ABB RAPID module: etna.mod

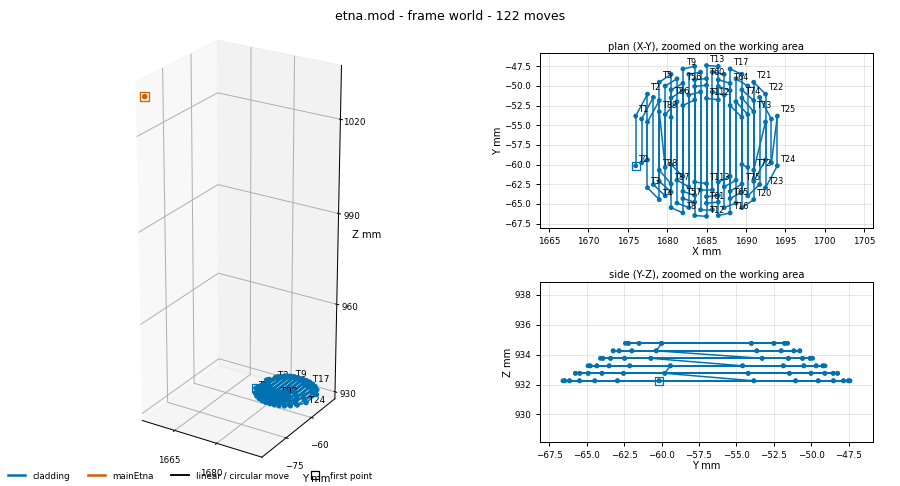
[picture p0: tool path of etna.mod in frame world, 122 of 122 moves have a stored position in this frame; points joined in program order, loops and branches not executed]
MODULE Etna

    PERS tooldata toolEtna:=[TRUE,[[215.7,-22.4,473.8],[0.500000,0.000000,-0.866025,0.000000]],[20,[70,30,123.5],[0,0,1,0],1,0,1]];
    PERS wobjdata wobjEtna:=[FALSE,TRUE,"",[[1655.0,-87.0,932.0],[1.000000,0.000000,0.000000,0.000000]],[[0,0,0],[1,0,0,0]]];

    VAR triggdata laserON;
    VAR triggdata laserOFF;

    CONST speeddata vl:=[8,500,5000,1000];


    CONST robtarget T0:=[[21.000000,26.839411,0.250000],[1.000000,0.000000,0.000000,0.000000],[-1,0,-1,0],[9E+09,9E+09,9E+09,9E+09,9E+09,9E+09]];
    CONST robtarget T1:=[[21.000000,33.160593,0.250000],[1.000000,0.000000,0.000000,0.000000],[-1,0,-1,0],[9E+09,9E+09,9E+09,9E+09,9E+09,9E+09]];
    CONST robtarget T2:=[[22.500000,35.946596,0.250000],[1.000000,0.000000,0.000000,0.000000],[-1,0,-1,0],[9E+09,9E+09,9E+09,9E+09,9E+09,9E+09]];
    CONST robtarget T3:=[[22.500000,24.053408,0.250000],[1.000000,0.000000,0.000000,0.000000],[-1,0,-1,0],[9E+09,9E+09,9E+09,9E+09,9E+09,9E+09]];
    CONST robtarget T4:=[[24.000000,22.537615,0.250000],[1.000000,0.000000,0.000000,0.000000],[-1,0,-1,0],[9E+09,9E+09,9E+09,9E+09,9E+09,9E+09]];
    CONST robtarget T5:=[[24.000000,37.462389,0.250000],[1.000000,0.000000,0.000000,0.000000],[-1,0,-1,0],[9E+09,9E+09,9E+09,9E+09,9E+09,9E+09]];
    CONST robtarget T6:=[[25.500000,38.475702,0.250000],[1.000000,0.000000,0.000000,0.000000],[-1,0,-1,0],[9E+09,9E+09,9E+09,9E+09,9E+09,9E+09]];
    CONST robtarget T7:=[[25.500000,21.524301,0.250000],[1.000000,0.000000,0.000000,0.000000],[-1,0,-1,0],[9E+09,9E+09,9E+09,9E+09,9E+09,9E+09]];
    CONST robtarget T8:=[[27.000000,20.852779,0.250000],[1.000000,0.000000,0.000000,0.000000],[-1,0,-1,0],[9E+09,9E+09,9E+09,9E+09,9E+09,9E+09]];
    CONST robtarget T9:=[[27.000000,39.147225,0.250000],[1.000000,0.000000,0.000000,0.000000],[-1,0,-1,0],[9E+09,9E+09,9E+09,9E+09,9E+09,9E+09]];
    CONST robtarget T10:=[[28.500000,39.476842,0.250000],[1.000000,0.000000,0.000000,0.000000],[-1,0,-1,0],[9E+09,9E+09,9E+09,9E+09,9E+09,9E+09]];
    CONST robtarget T11:=[[28.500000,20.523160,0.250000],[1.000000,0.000000,0.000000,0.000000],[-1,0,-1,0],[9E+09,9E+09,9E+09,9E+09,9E+09,9E+09]];
    CONST robtarget T12:=[[30.000000,20.416667,0.250000],[1.000000,0.000000,0.000000,0.000000],[-1,0,-1,0],[9E+09,9E+09,9E+09,9E+09,9E+09,9E+09]];
    CONST robtarget T13:=[[30.000000,39.583335,0.250000],[1.000000,0.000000,0.000000,0.000000],[-1,0,-1,0],[9E+09,9E+09,9E+09,9E+09,9E+09,9E+09]];
    CONST robtarget T14:=[[31.500000,39.476842,0.250000],[1.000000,0.000000,0.000000,0.000000],[-1,0,-1,0],[9E+09,9E+09,9E+09,9E+09,9E+09,9E+09]];
    CONST robtarget T15:=[[31.500000,20.523161,0.250000],[1.000000,0.000000,0.000000,0.000000],[-1,0,-1,0],[9E+09,9E+09,9E+09,9E+09,9E+09,9E+09]];
    CONST robtarget T16:=[[33.000000,20.852779,0.250000],[1.000000,0.000000,0.000000,0.000000],[-1,0,-1,0],[9E+09,9E+09,9E+09,9E+09,9E+09,9E+09]];
    CONST robtarget T17:=[[33.000000,39.147225,0.250000],[1.000000,0.000000,0.000000,0.000000],[-1,0,-1,0],[9E+09,9E+09,9E+09,9E+09,9E+09,9E+09]];
    CONST robtarget T18:=[[34.500000,38.475702,0.250000],[1.000000,0.000000,0.000000,0.000000],[-1,0,-1,0],[9E+09,9E+09,9E+09,9E+09,9E+09,9E+09]];
    CONST robtarget T19:=[[34.500000,21.524301,0.250000],[1.000000,0.000000,0.000000,0.000000],[-1,0,-1,0],[9E+09,9E+09,9E+09,9E+09,9E+09,9E+09]];
    CONST robtarget T20:=[[36.000000,22.537615,0.250000],[1.000000,0.000000,0.000000,0.000000],[-1,0,-1,0],[9E+09,9E+09,9E+09,9E+09,9E+09,9E+09]];
    CONST robtarget T21:=[[36.000000,37.462389,0.250000],[1.000000,0.000000,0.000000,0.000000],[-1,0,-1,0],[9E+09,9E+09,9E+09,9E+09,9E+09,9E+09]];
    CONST robtarget T22:=[[37.500000,35.946596,0.250000],[1.000000,0.000000,0.000000,0.000000],[-1,0,-1,0],[9E+09,9E+09,9E+09,9E+09,9E+09,9E+09]];
    CONST robtarget T23:=[[37.500000,24.053407,0.250000],[1.000000,0.000000,0.000000,0.000000],[-1,0,-1,0],[9E+09,9E+09,9E+09,9E+09,9E+09,9E+09]];
    CONST robtarget T24:=[[39.000000,26.839410,0.250000],[1.000000,0.000000,0.000000,0.000000],[-1,0,-1,0],[9E+09,9E+09,9E+09,9E+09,9E+09,9E+09]];
    CONST robtarget T25:=[[39.000000,33.160593,0.250000],[1.000000,0.000000,0.000000,0.000000],[-1,0,-1,0],[9E+09,9E+09,9E+09,9E+09,9E+09,9E+09]];
    CONST robtarget T26:=[[38.250000,27.215156,0.750000],[1.000000,0.000000,0.000000,0.000000],[-1,0,-1,0],[9E+09,9E+09,9E+09,9E+09,9E+09,9E+09]];
    CONST robtarget T27:=[[38.250000,32.784847,0.750000],[1.000000,0.000000,0.000000,0.000000],[-1,0,-1,0],[9E+09,9E+09,9E+09,9E+09,9E+09,9E+09]];
    CONST robtarget T28:=[[36.750000,35.538746,0.750000],[1.000000,0.000000,0.000000,0.000000],[-1,0,-1,0],[9E+09,9E+09,9E+09,9E+09,9E+09,9E+09]];
    CONST robtarget T29:=[[36.750000,24.461257,0.750000],[1.000000,0.000000,0.000000,0.000000],[-1,0,-1,0],[9E+09,9E+09,9E+09,9E+09,9E+09,9E+09]];
    CONST robtarget T30:=[[35.250000,23.019764,0.750000],[1.000000,0.000000,0.000000,0.000000],[-1,0,-1,0],[9E+09,9E+09,9E+09,9E+09,9E+09,9E+09]];
    CONST robtarget T31:=[[35.250000,36.980240,0.750000],[1.000000,0.000000,0.000000,0.000000],[-1,0,-1,0],[9E+09,9E+09,9E+09,9E+09,9E+09,9E+09]];
    CONST robtarget T32:=[[33.750000,37.899267,0.750000],[1.000000,0.000000,0.000000,0.000000],[-1,0,-1,0],[9E+09,9E+09,9E+09,9E+09,9E+09,9E+09]];
    CONST robtarget T33:=[[33.750000,22.100737,0.750000],[1.000000,0.000000,0.000000,0.000000],[-1,0,-1,0],[9E+09,9E+09,9E+09,9E+09,9E+09,9E+09]];
    CONST robtarget T34:=[[32.250000,21.535407,0.750000],[1.000000,0.000000,0.000000,0.000000],[-1,0,-1,0],[9E+09,9E+09,9E+09,9E+09,9E+09,9E+09]];
    CONST robtarget T35:=[[32.250000,38.464597,0.750000],[1.000000,0.000000,0.000000,0.000000],[-1,0,-1,0],[9E+09,9E+09,9E+09,9E+09,9E+09,9E+09]];
    CONST robtarget T36:=[[30.750000,38.750002,0.750000],[1.000000,0.000000,0.000000,0.000000],[-1,0,-1,0],[9E+09,9E+09,9E+09,9E+09,9E+09,9E+09]];
    CONST robtarget T37:=[[30.750000,21.250000,0.750000],[1.000000,0.000000,0.000000,0.000000],[-1,0,-1,0],[9E+09,9E+09,9E+09,9E+09,9E+09,9E+09]];
    CONST robtarget T38:=[[29.250000,21.250000,0.750000],[1.000000,0.000000,0.000000,0.000000],[-1,0,-1,0],[9E+09,9E+09,9E+09,9E+09,9E+09,9E+09]];
    CONST robtarget T39:=[[29.250000,38.750002,0.750000],[1.000000,0.000000,0.000000,0.000000],[-1,0,-1,0],[9E+09,9E+09,9E+09,9E+09,9E+09,9E+09]];
    CONST robtarget T40:=[[27.750000,38.464597,0.750000],[1.000000,0.000000,0.000000,0.000000],[-1,0,-1,0],[9E+09,9E+09,9E+09,9E+09,9E+09,9E+09]];
    CONST robtarget T41:=[[27.750000,21.535406,0.750000],[1.000000,0.000000,0.000000,0.000000],[-1,0,-1,0],[9E+09,9E+09,9E+09,9E+09,9E+09,9E+09]];
    CONST robtarget T42:=[[26.250000,22.100737,0.750000],[1.000000,0.000000,0.000000,0.000000],[-1,0,-1,0],[9E+09,9E+09,9E+09,9E+09,9E+09,9E+09]];
    CONST robtarget T43:=[[26.250000,37.899267,0.750000],[1.000000,0.000000,0.000000,0.000000],[-1,0,-1,0],[9E+09,9E+09,9E+09,9E+09,9E+09,9E+09]];
    CONST robtarget T44:=[[24.750000,36.980240,0.750000],[1.000000,0.000000,0.000000,0.000000],[-1,0,-1,0],[9E+09,9E+09,9E+09,9E+09,9E+09,9E+09]];
    CONST robtarget T45:=[[24.750000,23.019764,0.750000],[1.000000,0.000000,0.000000,0.000000],[-1,0,-1,0],[9E+09,9E+09,9E+09,9E+09,9E+09,9E+09]];
    CONST robtarget T46:=[[23.250000,24.461257,0.750000],[1.000000,0.000000,0.000000,0.000000],[-1,0,-1,0],[9E+09,9E+09,9E+09,9E+09,9E+09,9E+09]];
    CONST robtarget T47:=[[23.250000,35.538747,0.750000],[1.000000,0.000000,0.000000,0.000000],[-1,0,-1,0],[9E+09,9E+09,9E+09,9E+09,9E+09,9E+09]];
    CONST robtarget T48:=[[21.750000,32.784848,0.750000],[1.000000,0.000000,0.000000,0.000000],[-1,0,-1,0],[9E+09,9E+09,9E+09,9E+09,9E+09,9E+09]];
    CONST robtarget T49:=[[21.750000,27.215157,0.750000],[1.000000,0.000000,0.000000,0.000000],[-1,0,-1,0],[9E+09,9E+09,9E+09,9E+09,9E+09,9E+09]];
    CONST robtarget T50:=[[22.500000,27.590903,1.250000],[1.000000,0.000000,0.000000,0.000000],[-1,0,-1,0],[9E+09,9E+09,9E+09,9E+09,9E+09,9E+09]];
    CONST robtarget T51:=[[22.500000,32.409103,1.250000],[1.000000,0.000000,0.000000,0.000000],[-1,0,-1,0],[9E+09,9E+09,9E+09,9E+09,9E+09,9E+09]];
    CONST robtarget T52:=[[24.000000,35.130897,1.250000],[1.000000,0.000000,0.000000,0.000000],[-1,0,-1,0],[9E+09,9E+09,9E+09,9E+09,9E+09,9E+09]];
    CONST robtarget T53:=[[24.000000,24.869107,1.250000],[1.000000,0.000000,0.000000,0.000000],[-1,0,-1,0],[9E+09,9E+09,9E+09,9E+09,9E+09,9E+09]];
    CONST robtarget T54:=[[25.500000,23.501912,1.250000],[1.000000,0.000000,0.000000,0.000000],[-1,0,-1,0],[9E+09,9E+09,9E+09,9E+09,9E+09,9E+09]];
    CONST robtarget T55:=[[25.500000,36.498092,1.250000],[1.000000,0.000000,0.000000,0.000000],[-1,0,-1,0],[9E+09,9E+09,9E+09,9E+09,9E+09,9E+09]];
    CONST robtarget T56:=[[27.000000,37.322831,1.250000],[1.000000,0.000000,0.000000,0.000000],[-1,0,-1,0],[9E+09,9E+09,9E+09,9E+09,9E+09,9E+09]];
    CONST robtarget T57:=[[27.000000,22.677173,1.250000],[1.000000,0.000000,0.000000,0.000000],[-1,0,-1,0],[9E+09,9E+09,9E+09,9E+09,9E+09,9E+09]];
    CONST robtarget T58:=[[28.500000,22.227061,1.250000],[1.000000,0.000000,0.000000,0.000000],[-1,0,-1,0],[9E+09,9E+09,9E+09,9E+09,9E+09,9E+09]];
    CONST robtarget T59:=[[28.500000,37.772941,1.250000],[1.000000,0.000000,0.000000,0.000000],[-1,0,-1,0],[9E+09,9E+09,9E+09,9E+09,9E+09,9E+09]];
    CONST robtarget T60:=[[30.000000,37.916669,1.250000],[1.000000,0.000000,0.000000,0.000000],[-1,0,-1,0],[9E+09,9E+09,9E+09,9E+09,9E+09,9E+09]];
    CONST robtarget T61:=[[30.000000,22.083334,1.250000],[1.000000,0.000000,0.000000,0.000000],[-1,0,-1,0],[9E+09,9E+09,9E+09,9E+09,9E+09,9E+09]];
    CONST robtarget T62:=[[31.500000,22.227062,1.250000],[1.000000,0.000000,0.000000,0.000000],[-1,0,-1,0],[9E+09,9E+09,9E+09,9E+09,9E+09,9E+09]];
    CONST robtarget T63:=[[31.500000,37.772942,1.250000],[1.000000,0.000000,0.000000,0.000000],[-1,0,-1,0],[9E+09,9E+09,9E+09,9E+09,9E+09,9E+09]];
    CONST robtarget T64:=[[33.000000,37.322831,1.250000],[1.000000,0.000000,0.000000,0.000000],[-1,0,-1,0],[9E+09,9E+09,9E+09,9E+09,9E+09,9E+09]];
    CONST robtarget T65:=[[33.000000,22.677173,1.250000],[1.000000,0.000000,0.000000,0.000000],[-1,0,-1,0],[9E+09,9E+09,9E+09,9E+09,9E+09,9E+09]];
    CONST robtarget T66:=[[34.500000,23.501912,1.250000],[1.000000,0.000000,0.000000,0.000000],[-1,0,-1,0],[9E+09,9E+09,9E+09,9E+09,9E+09,9E+09]];
    CONST robtarget T67:=[[34.500000,36.498092,1.250000],[1.000000,0.000000,0.000000,0.000000],[-1,0,-1,0],[9E+09,9E+09,9E+09,9E+09,9E+09,9E+09]];
    CONST robtarget T68:=[[36.000000,35.130896,1.250000],[1.000000,0.000000,0.000000,0.000000],[-1,0,-1,0],[9E+09,9E+09,9E+09,9E+09,9E+09,9E+09]];
    CONST robtarget T69:=[[36.000000,24.869107,1.250000],[1.000000,0.000000,0.000000,0.000000],[-1,0,-1,0],[9E+09,9E+09,9E+09,9E+09,9E+09,9E+09]];
    CONST robtarget T70:=[[37.500000,27.590901,1.250000],[1.000000,0.000000,0.000000,0.000000],[-1,0,-1,0],[9E+09,9E+09,9E+09,9E+09,9E+09,9E+09]];
    CONST robtarget T71:=[[37.500000,32.409101,1.250000],[1.000000,0.000000,0.000000,0.000000],[-1,0,-1,0],[9E+09,9E+09,9E+09,9E+09,9E+09,9E+09]];
    CONST robtarget T72:=[[36.000000,26.282882,1.750000],[1.000000,0.000000,0.000000,0.000000],[-1,0,-1,0],[9E+09,9E+09,9E+09,9E+09,9E+09,9E+09]];
    CONST robtarget T73:=[[36.000000,33.717123,1.750000],[1.000000,0.000000,0.000000,0.000000],[-1,0,-1,0],[9E+09,9E+09,9E+09,9E+09,9E+09,9E+09]];
    CONST robtarget T74:=[[34.500000,35.468036,1.750000],[1.000000,0.000000,0.000000,0.000000],[-1,0,-1,0],[9E+09,9E+09,9E+09,9E+09,9E+09,9E+09]];
    CONST robtarget T75:=[[34.500000,24.531968,1.750000],[1.000000,0.000000,0.000000,0.000000],[-1,0,-1,0],[9E+09,9E+09,9E+09,9E+09,9E+09,9E+09]];
    CONST robtarget T76:=[[33.000000,23.589370,1.750000],[1.000000,0.000000,0.000000,0.000000],[-1,0,-1,0],[9E+09,9E+09,9E+09,9E+09,9E+09,9E+09]];
    CONST robtarget T77:=[[33.000000,36.410634,1.750000],[1.000000,0.000000,0.000000,0.000000],[-1,0,-1,0],[9E+09,9E+09,9E+09,9E+09,9E+09,9E+09]];
    CONST robtarget T78:=[[31.500000,36.920992,1.750000],[1.000000,0.000000,0.000000,0.000000],[-1,0,-1,0],[9E+09,9E+09,9E+09,9E+09,9E+09,9E+09]];
    CONST robtarget T79:=[[31.500000,23.079013,1.750000],[1.000000,0.000000,0.000000,0.000000],[-1,0,-1,0],[9E+09,9E+09,9E+09,9E+09,9E+09,9E+09]];
    CONST robtarget T80:=[[30.000000,22.916668,1.750000],[1.000000,0.000000,0.000000,0.000000],[-1,0,-1,0],[9E+09,9E+09,9E+09,9E+09,9E+09,9E+09]];
    CONST robtarget T81:=[[30.000000,37.083335,1.750000],[1.000000,0.000000,0.000000,0.000000],[-1,0,-1,0],[9E+09,9E+09,9E+09,9E+09,9E+09,9E+09]];
    CONST robtarget T82:=[[28.500000,36.920991,1.750000],[1.000000,0.000000,0.000000,0.000000],[-1,0,-1,0],[9E+09,9E+09,9E+09,9E+09,9E+09,9E+09]];
    CONST robtarget T83:=[[28.500000,23.079011,1.750000],[1.000000,0.000000,0.000000,0.000000],[-1,0,-1,0],[9E+09,9E+09,9E+09,9E+09,9E+09,9E+09]];
    CONST robtarget T84:=[[27.000000,23.589370,1.750000],[1.000000,0.000000,0.000000,0.000000],[-1,0,-1,0],[9E+09,9E+09,9E+09,9E+09,9E+09,9E+09]];
    CONST robtarget T85:=[[27.000000,36.410634,1.750000],[1.000000,0.000000,0.000000,0.000000],[-1,0,-1,0],[9E+09,9E+09,9E+09,9E+09,9E+09,9E+09]];
    CONST robtarget T86:=[[25.500000,35.468036,1.750000],[1.000000,0.000000,0.000000,0.000000],[-1,0,-1,0],[9E+09,9E+09,9E+09,9E+09,9E+09,9E+09]];
    CONST robtarget T87:=[[25.500000,24.531968,1.750000],[1.000000,0.000000,0.000000,0.000000],[-1,0,-1,0],[9E+09,9E+09,9E+09,9E+09,9E+09,9E+09]];
    CONST robtarget T88:=[[24.000000,26.282881,1.750000],[1.000000,0.000000,0.000000,0.000000],[-1,0,-1,0],[9E+09,9E+09,9E+09,9E+09,9E+09,9E+09]];
    CONST robtarget T89:=[[24.000000,33.717121,1.750000],[1.000000,0.000000,0.000000,0.000000],[-1,0,-1,0],[9E+09,9E+09,9E+09,9E+09,9E+09,9E+09]];
    CONST robtarget T90:=[[24.750000,26.643354,2.250000],[1.000000,0.000000,0.000000,0.000000],[-1,0,-1,0],[9E+09,9E+09,9E+09,9E+09,9E+09,9E+09]];
    CONST robtarget T91:=[[24.750000,33.356648,2.250000],[1.000000,0.000000,0.000000,0.000000],[-1,0,-1,0],[9E+09,9E+09,9E+09,9E+09,9E+09,9E+09]];
    CONST robtarget T92:=[[26.250000,34.985887,2.250000],[1.000000,0.000000,0.000000,0.000000],[-1,0,-1,0],[9E+09,9E+09,9E+09,9E+09,9E+09,9E+09]];
    CONST robtarget T93:=[[26.250000,25.014116,2.250000],[1.000000,0.000000,0.000000,0.000000],[-1,0,-1,0],[9E+09,9E+09,9E+09,9E+09,9E+09,9E+09]];
    CONST robtarget T94:=[[27.750000,24.165805,2.250000],[1.000000,0.000000,0.000000,0.000000],[-1,0,-1,0],[9E+09,9E+09,9E+09,9E+09,9E+09,9E+09]];
    CONST robtarget T95:=[[27.750000,35.834199,2.250000],[1.000000,0.000000,0.000000,0.000000],[-1,0,-1,0],[9E+09,9E+09,9E+09,9E+09,9E+09,9E+09]];
    CONST robtarget T96:=[[29.250000,36.229335,2.250000],[1.000000,0.000000,0.000000,0.000000],[-1,0,-1,0],[9E+09,9E+09,9E+09,9E+09,9E+09,9E+09]];
    CONST robtarget T97:=[[29.250000,23.770668,2.250000],[1.000000,0.000000,0.000000,0.000000],[-1,0,-1,0],[9E+09,9E+09,9E+09,9E+09,9E+09,9E+09]];
    CONST robtarget T98:=[[30.750000,23.770668,2.250000],[1.000000,0.000000,0.000000,0.000000],[-1,0,-1,0],[9E+09,9E+09,9E+09,9E+09,9E+09,9E+09]];
    CONST robtarget T99:=[[30.750000,36.229335,2.250000],[1.000000,0.000000,0.000000,0.000000],[-1,0,-1,0],[9E+09,9E+09,9E+09,9E+09,9E+09,9E+09]];
    CONST robtarget T100:=[[32.250000,35.834199,2.250000],[1.000000,0.000000,0.000000,0.000000],[-1,0,-1,0],[9E+09,9E+09,9E+09,9E+09,9E+09,9E+09]];
    CONST robtarget T101:=[[32.250000,24.165805,2.250000],[1.000000,0.000000,0.000000,0.000000],[-1,0,-1,0],[9E+09,9E+09,9E+09,9E+09,9E+09,9E+09]];
    CONST robtarget T102:=[[33.750000,25.014116,2.250000],[1.000000,0.000000,0.000000,0.000000],[-1,0,-1,0],[9E+09,9E+09,9E+09,9E+09,9E+09,9E+09]];
    CONST robtarget T103:=[[33.750000,34.985887,2.250000],[1.000000,0.000000,0.000000,0.000000],[-1,0,-1,0],[9E+09,9E+09,9E+09,9E+09,9E+09,9E+09]];
    CONST robtarget T104:=[[35.250000,33.356650,2.250000],[1.000000,0.000000,0.000000,0.000000],[-1,0,-1,0],[9E+09,9E+09,9E+09,9E+09,9E+09,9E+09]];
    CONST robtarget T105:=[[35.250000,26.643356,2.250000],[1.000000,0.000000,0.000000,0.000000],[-1,0,-1,0],[9E+09,9E+09,9E+09,9E+09,9E+09,9E+09]];
    CONST robtarget T106:=[[34.500000,27.003828,2.750000],[1.000000,0.000000,0.000000,0.000000],[-1,0,-1,0],[9E+09,9E+09,9E+09,9E+09,9E+09,9E+09]];
    CONST robtarget T107:=[[34.500000,32.996176,2.750000],[1.000000,0.000000,0.000000,0.000000],[-1,0,-1,0],[9E+09,9E+09,9E+09,9E+09,9E+09,9E+09]];
    CONST robtarget T108:=[[33.000000,34.503739,2.750000],[1.000000,0.000000,0.000000,0.000000],[-1,0,-1,0],[9E+09,9E+09,9E+09,9E+09,9E+09,9E+09]];
    CONST robtarget T109:=[[33.000000,25.496265,2.750000],[1.000000,0.000000,0.000000,0.000000],[-1,0,-1,0],[9E+09,9E+09,9E+09,9E+09,9E+09,9E+09]];
    CONST robtarget T110:=[[31.500000,24.782912,2.750000],[1.000000,0.000000,0.000000,0.000000],[-1,0,-1,0],[9E+09,9E+09,9E+09,9E+09,9E+09,9E+09]];
    CONST robtarget T111:=[[31.500000,35.217092,2.750000],[1.000000,0.000000,0.000000,0.000000],[-1,0,-1,0],[9E+09,9E+09,9E+09,9E+09,9E+09,9E+09]];
    CONST robtarget T112:=[[30.000000,35.416669,2.750000],[1.000000,0.000000,0.000000,0.000000],[-1,0,-1,0],[9E+09,9E+09,9E+09,9E+09,9E+09,9E+09]];
    CONST robtarget T113:=[[30.000000,24.583335,2.750000],[1.000000,0.000000,0.000000,0.000000],[-1,0,-1,0],[9E+09,9E+09,9E+09,9E+09,9E+09,9E+09]];
    CONST robtarget T114:=[[28.500000,24.782912,2.750000],[1.000000,0.000000,0.000000,0.000000],[-1,0,-1,0],[9E+09,9E+09,9E+09,9E+09,9E+09,9E+09]];
    CONST robtarget T115:=[[28.500000,35.217091,2.750000],[1.000000,0.000000,0.000000,0.000000],[-1,0,-1,0],[9E+09,9E+09,9E+09,9E+09,9E+09,9E+09]];
    CONST robtarget T116:=[[27.000000,34.503739,2.750000],[1.000000,0.000000,0.000000,0.000000],[-1,0,-1,0],[9E+09,9E+09,9E+09,9E+09,9E+09,9E+09]];
    CONST robtarget T117:=[[27.000000,25.496265,2.750000],[1.000000,0.000000,0.000000,0.000000],[-1,0,-1,0],[9E+09,9E+09,9E+09,9E+09,9E+09,9E+09]];
    CONST robtarget T118:=[[25.500000,27.003828,2.750000],[1.000000,0.000000,0.000000,0.000000],[-1,0,-1,0],[9E+09,9E+09,9E+09,9E+09,9E+09,9E+09]];
    CONST robtarget T119:=[[25.500000,32.996175,2.750000],[1.000000,0.000000,0.000000,0.000000],[-1,0,-1,0],[9E+09,9E+09,9E+09,9E+09,9E+09,9E+09]];

PROC cladding()
    !Reset doLDLStartST;

    TriggL T0,v50,laserON,z0,toolEtna\WObj:=wobjEtna;
    TriggL T1,vl,laserOFF,z0,toolEtna\WObj:=wobjEtna;
    TriggL T2,v50,laserON,z0,toolEtna\WObj:=wobjEtna;
    TriggL T3,vl,laserOFF,z0,toolEtna\WObj:=wobjEtna;
    TriggL T4,v50,laserON,z0,toolEtna\WObj:=wobjEtna;
    TriggL T5,vl,laserOFF,z0,toolEtna\WObj:=wobjEtna;
    TriggL T6,v50,laserON,z0,toolEtna\WObj:=wobjEtna;
    TriggL T7,vl,laserOFF,z0,toolEtna\WObj:=wobjEtna;
    TriggL T8,v50,laserON,z0,toolEtna\WObj:=wobjEtna;
    TriggL T9,vl,laserOFF,z0,toolEtna\WObj:=wobjEtna;
    TriggL T10,v50,laserON,z0,toolEtna\WObj:=wobjEtna;
    TriggL T11,vl,laserOFF,z0,toolEtna\WObj:=wobjEtna;
    TriggL T12,v50,laserON,z0,toolEtna\WObj:=wobjEtna;
    TriggL T13,vl,laserOFF,z0,toolEtna\WObj:=wobjEtna;
    TriggL T14,v50,laserON,z0,toolEtna\WObj:=wobjEtna;
    TriggL T15,vl,laserOFF,z0,toolEtna\WObj:=wobjEtna;
    TriggL T16,v50,laserON,z0,toolEtna\WObj:=wobjEtna;
    TriggL T17,vl,laserOFF,z0,toolEtna\WObj:=wobjEtna;
    TriggL T18,v50,laserON,z0,toolEtna\WObj:=wobjEtna;
    TriggL T19,vl,laserOFF,z0,toolEtna\WObj:=wobjEtna;
    TriggL T20,v50,laserON,z0,toolEtna\WObj:=wobjEtna;
    TriggL T21,vl,laserOFF,z0,toolEtna\WObj:=wobjEtna;
    TriggL T22,v50,laserON,z0,toolEtna\WObj:=wobjEtna;
    TriggL T23,vl,laserOFF,z0,toolEtna\WObj:=wobjEtna;
    TriggL T24,v50,laserON,z0,toolEtna\WObj:=wobjEtna;
    TriggL T25,vl,laserOFF,z0,toolEtna\WObj:=wobjEtna;
    TriggL T26,v50,laserON,z0,toolEtna\WObj:=wobjEtna;
    TriggL T27,vl,laserOFF,z0,toolEtna\WObj:=wobjEtna;
    TriggL T28,v50,laserON,z0,toolEtna\WObj:=wobjEtna;
    TriggL T29,vl,laserOFF,z0,toolEtna\WObj:=wobjEtna;
    TriggL T30,v50,laserON,z0,toolEtna\WObj:=wobjEtna;
    TriggL T31,vl,laserOFF,z0,toolEtna\WObj:=wobjEtna;
    TriggL T32,v50,laserON,z0,toolEtna\WObj:=wobjEtna;
    TriggL T33,vl,laserOFF,z0,toolEtna\WObj:=wobjEtna;
    TriggL T34,v50,laserON,z0,toolEtna\WObj:=wobjEtna;
    TriggL T35,vl,laserOFF,z0,toolEtna\WObj:=wobjEtna;
    TriggL T36,v50,laserON,z0,toolEtna\WObj:=wobjEtna;
    TriggL T37,vl,laserOFF,z0,toolEtna\WObj:=wobjEtna;
    TriggL T38,v50,laserON,z0,toolEtna\WObj:=wobjEtna;
    TriggL T39,vl,laserOFF,z0,toolEtna\WObj:=wobjEtna;
    TriggL T40,v50,laserON,z0,toolEtna\WObj:=wobjEtna;
    TriggL T41,vl,laserOFF,z0,toolEtna\WObj:=wobjEtna;
    TriggL T42,v50,laserON,z0,toolEtna\WObj:=wobjEtna;
    TriggL T43,vl,laserOFF,z0,toolEtna\WObj:=wobjEtna;
    TriggL T44,v50,laserON,z0,toolEtna\WObj:=wobjEtna;
    TriggL T45,vl,laserOFF,z0,toolEtna\WObj:=wobjEtna;
    TriggL T46,v50,laserON,z0,toolEtna\WObj:=wobjEtna;
    TriggL T47,vl,laserOFF,z0,toolEtna\WObj:=wobjEtna;
    TriggL T48,v50,laserON,z0,toolEtna\WObj:=wobjEtna;
    TriggL T49,vl,laserOFF,z0,toolEtna\WObj:=wobjEtna;
    TriggL T50,v50,laserON,z0,toolEtna\WObj:=wobjEtna;
    TriggL T51,vl,laserOFF,z0,toolEtna\WObj:=wobjEtna;
    TriggL T52,v50,laserON,z0,toolEtna\WObj:=wobjEtna;
    TriggL T53,vl,laserOFF,z0,toolEtna\WObj:=wobjEtna;
    TriggL T54,v50,laserON,z0,toolEtna\WObj:=wobjEtna;
    TriggL T55,vl,laserOFF,z0,toolEtna\WObj:=wobjEtna;
    TriggL T56,v50,laserON,z0,toolEtna\WObj:=wobjEtna;
    TriggL T57,vl,laserOFF,z0,toolEtna\WObj:=wobjEtna;
    TriggL T58,v50,laserON,z0,toolEtna\WObj:=wobjEtna;
    TriggL T59,vl,laserOFF,z0,toolEtna\WObj:=wobjEtna;
    TriggL T60,v50,laserON,z0,toolEtna\WObj:=wobjEtna;
    TriggL T61,vl,laserOFF,z0,toolEtna\WObj:=wobjEtna;
    TriggL T62,v50,laserON,z0,toolEtna\WObj:=wobjEtna;
    TriggL T63,vl,laserOFF,z0,toolEtna\WObj:=wobjEtna;
    TriggL T64,v50,laserON,z0,toolEtna\WObj:=wobjEtna;
    TriggL T65,vl,laserOFF,z0,toolEtna\WObj:=wobjEtna;
    TriggL T66,v50,laserON,z0,toolEtna\WObj:=wobjEtna;
    TriggL T67,vl,laserOFF,z0,toolEtna\WObj:=wobjEtna;
    TriggL T68,v50,laserON,z0,toolEtna\WObj:=wobjEtna;
    TriggL T69,vl,laserOFF,z0,toolEtna\WObj:=wobjEtna;
    TriggL T70,v50,laserON,z0,toolEtna\WObj:=wobjEtna;
    TriggL T71,vl,laserOFF,z0,toolEtna\WObj:=wobjEtna;
    TriggL T72,v50,laserON,z0,toolEtna\WObj:=wobjEtna;
    TriggL T73,vl,laserOFF,z0,toolEtna\WObj:=wobjEtna;
    TriggL T74,v50,laserON,z0,toolEtna\WObj:=wobjEtna;
    TriggL T75,vl,laserOFF,z0,toolEtna\WObj:=wobjEtna;
    TriggL T76,v50,laserON,z0,toolEtna\WObj:=wobjEtna;
    TriggL T77,vl,laserOFF,z0,toolEtna\WObj:=wobjEtna;
    TriggL T78,v50,laserON,z0,toolEtna\WObj:=wobjEtna;
    TriggL T79,vl,laserOFF,z0,toolEtna\WObj:=wobjEtna;
    TriggL T80,v50,laserON,z0,toolEtna\WObj:=wobjEtna;
    TriggL T81,vl,laserOFF,z0,toolEtna\WObj:=wobjEtna;
    TriggL T82,v50,laserON,z0,toolEtna\WObj:=wobjEtna;
    TriggL T83,vl,laserOFF,z0,toolEtna\WObj:=wobjEtna;
    TriggL T84,v50,laserON,z0,toolEtna\WObj:=wobjEtna;
    TriggL T85,vl,laserOFF,z0,toolEtna\WObj:=wobjEtna;
    TriggL T86,v50,laserON,z0,toolEtna\WObj:=wobjEtna;
    TriggL T87,vl,laserOFF,z0,toolEtna\WObj:=wobjEtna;
    TriggL T88,v50,laserON,z0,toolEtna\WObj:=wobjEtna;
    TriggL T89,vl,laserOFF,z0,toolEtna\WObj:=wobjEtna;
    TriggL T90,v50,laserON,z0,toolEtna\WObj:=wobjEtna;
    TriggL T91,vl,laserOFF,z0,toolEtna\WObj:=wobjEtna;
    TriggL T92,v50,laserON,z0,toolEtna\WObj:=wobjEtna;
    TriggL T93,vl,laserOFF,z0,toolEtna\WObj:=wobjEtna;
    TriggL T94,v50,laserON,z0,toolEtna\WObj:=wobjEtna;
    TriggL T95,vl,laserOFF,z0,toolEtna\WObj:=wobjEtna;
    TriggL T96,v50,laserON,z0,toolEtna\WObj:=wobjEtna;
    TriggL T97,vl,laserOFF,z0,toolEtna\WObj:=wobjEtna;
    TriggL T98,v50,laserON,z0,toolEtna\WObj:=wobjEtna;
    TriggL T99,vl,laserOFF,z0,toolEtna\WObj:=wobjEtna;
    TriggL T100,v50,laserON,z0,toolEtna\WObj:=wobjEtna;
    TriggL T101,vl,laserOFF,z0,toolEtna\WObj:=wobjEtna;
    TriggL T102,v50,laserON,z0,toolEtna\WObj:=wobjEtna;
    TriggL T103,vl,laserOFF,z0,toolEtna\WObj:=wobjEtna;
    TriggL T104,v50,laserON,z0,toolEtna\WObj:=wobjEtna;
    TriggL T105,vl,laserOFF,z0,toolEtna\WObj:=wobjEtna;
    TriggL T106,v50,laserON,z0,toolEtna\WObj:=wobjEtna;
    TriggL T107,vl,laserOFF,z0,toolEtna\WObj:=wobjEtna;
    TriggL T108,v50,laserON,z0,toolEtna\WObj:=wobjEtna;
    TriggL T109,vl,laserOFF,z0,toolEtna\WObj:=wobjEtna;
    TriggL T110,v50,laserON,z0,toolEtna\WObj:=wobjEtna;
    TriggL T111,vl,laserOFF,z0,toolEtna\WObj:=wobjEtna;
    TriggL T112,v50,laserON,z0,toolEtna\WObj:=wobjEtna;
    TriggL T113,vl,laserOFF,z0,toolEtna\WObj:=wobjEtna;
    TriggL T114,v50,laserON,z0,toolEtna\WObj:=wobjEtna;
    TriggL T115,vl,laserOFF,z0,toolEtna\WObj:=wobjEtna;
    TriggL T116,v50,laserON,z0,toolEtna\WObj:=wobjEtna;
    TriggL T117,vl,laserOFF,z0,toolEtna\WObj:=wobjEtna;
    TriggL T118,v50,laserON,z0,toolEtna\WObj:=wobjEtna;
    TriggL T119,vl,laserOFF,z0,toolEtna\WObj:=wobjEtna;

!Reset doLDLStartST;
ENDPROC

PROC mainEtna()
    Set Do_RF_MainOn;
    Set Do_RF_StandByOn;
    WaitDI DI_RF_LaserBeamReady,1;
    WaitDI DI_RF_GeneralFault,0;

    SetGO GO_Program_Rf, 0;
    WaitTime 1;
    !SetGO GoLDL_Pwr3, 1200;

    TriggIO laserON, 0\DOp:=Do_RF_ExterGate, 1;
    TriggIO laserOFF, 0\DOp:=Do_RF_ExterGate, 0;

    Set DoWeldGas;
    !MedicoatL2 "OFF", 5, 20, 7.5;
    MedicoatL1 "OFF", 3, 20, 20;

    ConfL \Off;

    MoveL [[0.0,0.0,100.0],[1.0,0.0,0.0,0.0],[-1,0,-1,0],[9E+09,9E+09,9E+09,9E+09,9E+09,9E+09]],v80,z0,toolEtna\WObj:=wobjEtna;

    cladding;

    MoveL [[0.0,0.0,100.0],[1.0,0.0,0.0,0.0],[-1,0,-1,0],[9E+09,9E+09,9E+09,9E+09,9E+09,9E+09]],v80,z0,toolEtna\WObj:=wobjEtna;

    Reset doMdtPL2On;
    Reset doMdtPL1On;
    Reset DoWeldGas;

    Reset Do_RF_StandByOn;
    !Reset Do_RF_MainOn;

ENDPROC

ENDMODULE
